{attribute 'pack_mode' := '1'}
TYPE TRunDataTurnOver :
STRUCT
	aTPartData						: ARRAY[0..1] OF TPartData;
END_STRUCT
END_TYPE

(* stored: Version 1.1.0.1, ProductVersion 3.1.4022.12
   DUT TRunDataTurnOver: Id {4e98f1d2-2b36-4348-a0ad-ae1b731bb4aa} *)
